# EPICS substitutions: modules/SAI/SAIApp/Db/SAI_IOCsystem.substitutions
# DEVICE: device name
# CARD:
# CS_VERSION_VAL

file /opt/epics/modules/uIOCSystem/db/system.template {
pattern { DEVICE, CARD, CS_VERSION_VAL}
	{ "FMBSAIIOC01", "0", "testing" }
}

#EOF
